TYPE T_FSS_RejecCode : STRING(40);
END_TYPE

(* stored: Version 1.1.0.1, ProductVersion 3.1.4024.15
   DUT T_FSS_RejecCode: Id {edc672d4-f5fd-4471-958c-1d92fe2bbb81} *)
